PROGRAM PRG_MainChamber
VAR
	fb_MC_Y : FB_MotionStage;
	bInit : BOOL := FALSE;
END_VAR

IF ( bInit) THEN
    bInit := FALSE;
    Main.M1.bHardwareEnable := TRUE;
    Main.M1.bPowerSelf := TRUE;
    Main.M1.nBrakeMode := ENUM_StageBrakeMode.NO_BRAKE;
    Main.M1.nEnableMode := ENUM_StageEnableMode.DURING_MOTION;
    END_IF
	
fb_MC_Y(stMotionStage := Main.M1);

END_PROGRAM

(* stored: Version 1.1.0.1, ProductVersion 3.1.4022.18
   POU PRG_MainChamber: Id {44b5b2b4-40eb-49d4-bd3b-945290e559d8}, SpecialFunc None *)
